(* IEC 61131-3 sources: OpenPLC-Simulator/openplc/OpenPLC/src, 47 files *)

(* ---- types.st ---- *)
(* ============================================================
   types.st — Data type definitions for the transporter simulator
   ============================================================ *)

TYPE TANK_T :
STRUCT
  tank_id    : INT;
  status     : INT;    (* NOT_USED=0, USED=1 *)
  x_position : REAL;
  y_position : REAL;
  z_position : REAL;
  stn_type   : INT;
END_STRUCT;
END_TYPE

TYPE STATION_T :
STRUCT
  tank_id       : INT;
  status        : INT;    (* NOT_USED=0, USED=1 *)
  x_position    : REAL;
  y_position    : REAL;
  z_position    : REAL;
  stn_type      : INT;    (* 0=dry, 1=wet *)
  stn_function  : INT;    (* original station type from JSON *)
  dropping_time : REAL;
  device_delay  : REAL;
END_STRUCT;
END_TYPE

TYPE PHYSICS_2D_T :
STRUCT
  x_accel_s      : REAL;
  x_decel_s      : REAL;
  x_max_mm_s     : REAL;
  z_total_mm     : REAL;
  z_slow_dry_mm  : REAL;
  z_slow_wet_mm  : REAL;
  z_slow_end_mm  : REAL;
  z_slow_mm_s    : REAL;
  z_fast_mm_s    : REAL;
  drip_delay_s   : REAL;
  avoid_mm       : REAL;
END_STRUCT;
END_TYPE

TYPE TASK_AREA_T :
STRUCT
  min_lift : INT;
  max_lift : INT;
  min_sink : INT;
  max_sink : INT;
END_STRUCT;
END_TYPE

TYPE TRANSPORTER_CFG_T :
STRUCT
  x_min_limit : REAL;
  x_max_limit : REAL;
  y_min_limit : REAL;
  y_max_limit : REAL;
  x_avoid_mm  : REAL;
  y_avoid_mm  : REAL;
  phys2d      : PHYSICS_2D_T;
  task_area   : ARRAY[1..4] OF TASK_AREA_T;
END_STRUCT;
END_TYPE

(* ── Transporter interface — production-compatible ──────────── *)
(* Used by scheduler, TWA, simulation, and production alike.     *)
(* g_transporter : ARRAY[1..TRANSPORTERS] OF STC_TRANSPORTER_T              *)
TYPE STC_TRANSPORTER_T :
STRUCT
  (* --- Command (scheduler → transporter) --- *)
  task_id            : LINT;     (* g_time_s at assignment — sync key *)
  lift_station       : INT;      (* pickup station number *)
  sink_station       : INT;      (* putdown station number *)
  treatment_time     : REAL;     (* treatment duration (s) *)
  lift_device_delay  : REAL;     (* lift station device delay (s) *)
  sink_device_delay  : REAL;     (* sink station device delay (s) *)
  dropping_time      : REAL;     (* dripping/dropping time at lift (s) *)
  (* --- Status (transporter → outside world) --- *)
  status             : INT;      (* 0=not_used 1=manual 2=half_manual 3=auto_idle 4=auto_run *)
  phase              : INT;      (* 0=idle 1=to_lift 2=lifting 3=to_sink 4=sinking *)
  running_task_id    : LINT;     (* copied from task_id when accepted *)
  current_station    : INT;      (* nearest station number *)
  remaining_time     : REAL;     (* remaining treatment time (s) *)
  (* --- Drive (runtime / TWA) --- *)
  final_target_x     : REAL;     (* destination X (station position) *)
  drive_target_x     : REAL;     (* TWA-clamped X drive target *)
  final_target_y     : REAL;     (* destination Y (3D transporter) *)
  drive_target_y     : REAL;     (* TWA-clamped Y drive target *)
  x_mm               : REAL;     (* current X position *)
  y_mm               : REAL;     (* current Y position (3D) *)
  z_mm               : REAL;     (* current Z position *)
  vel_x              : REAL;     (* X velocity *)
  z_stage            : INT;      (* Z motion sub-phase *)
  z_timer_s          : REAL;     (* Z motion timer *)
  x_min_limit        : REAL;     (* TWA lower X limit *)
  x_max_limit        : REAL;     (* TWA upper X limit *)
  (* --- General --- *)
  active             : BOOL;     (* transporter enabled *)
END_STRUCT;
END_TYPE

TYPE BATCH_T :
STRUCT
  batch_code : INT;     (* numeric batch code, e.g. 1, 2, 3 *)
  state      : INT;     (* NOT_PROCESSED=0, IN_PROCESS=1, PROCESSED=2 *)
  prog_id    : INT;     (* treatment program number *)
  cur_stage  : INT;     (* current stage number, 0 = not started *)
END_STRUCT;
END_TYPE

TYPE PROGRAM_STAGE_T :
STRUCT
  stations : ARRAY[1..5] OF INT;   (* up to MAX_PARALLELS station numbers *)
  min_time : INT;                   (* minimum processing time (seconds) *)
  max_time : INT;                   (* maximum processing time (seconds) *)
  cal_time : INT;                   (* calculated / target time (seconds) *)
END_STRUCT;
END_TYPE

TYPE TREATMENT_PROGRAM_T :
STRUCT
  program_id : INT;                      (* treatment program number *)
  stages     : ARRAY[1..30] OF PROGRAM_STAGE_T;  (* up to MAX_STAGES *)
END_STRUCT;
END_TYPE

TYPE UNIT_T :
STRUCT
  location : INT;    (* station number where unit currently is *)
  status   : INT;    (* NOT_USED=0, USED=1 *)
  state    : INT;    (* EMPTY=0, FULL=1 *)
  target   : INT;    (* TO_NONE=0, TO_LOADING=1, TO_BUFFER=2, TO_PROCESS=3, TO_UNLOAD=4, TO_AVOID=5 *)
END_STRUCT;
END_TYPE

(* ── Task Scheduler types (TSK_) ─────────────────────────────────── *)
(* Calculated batch schedule — one per unit, stages indexed 1..30       *)
(* Times are absolute epoch-offset seconds (g_time_s reference frame)   *)
(* Access: g_schedule[unit].stages[stage].entry_time                    *)

TYPE TSK_STAGE_T :
STRUCT
  station       : INT;     (* station number, 0 = unused stage *)
  entry_time    : LINT;    (* absolute arrival time (s), unix seconds *)
  exit_time     : LINT;    (* absolute departure time (s), unix seconds *)
  min_time      : REAL;    (* minimum treatment time (s) *)
  calc_time     : REAL;    (* calculated target treatment time (s) *)
  max_time      : REAL;    (* maximum treatment time (s) *)
  transfer_time : REAL;    (* transfer time from previous station (s) *)
END_STRUCT;
END_TYPE

TYPE TSK_SCHEDULE_T :
STRUCT
  stage_count : INT;                              (* number of active stages *)
  stages      : ARRAY[1..30] OF TSK_STAGE_T;     (* MAX_STAGES *)
END_STRUCT;
END_TYPE

(* Transporter task queue — indexed by transporter, then task slot       *)
(* unit is direct index to g_batches, g_programs, g_schedule, g_units   *)
(* Access: g_tasks[transporter].queue[slot].lift_station                *)

TYPE TSK_TASK_T :
STRUCT
  unit         : INT;     (* unit index 1..10, 0 = no task *)
  stage        : INT;     (* program stage that created this task *)
  lift_station : INT;     (* station to pick up from *)
  sink_station : INT;     (* station to put down to *)
  start_time   : LINT;    (* absolute time task begins (s), unix seconds *)
  finish_time  : LINT;    (* absolute time task completes (s), unix seconds *)
  calc_time    : REAL;    (* treatment calc_time for flex (s) *)
  min_time     : REAL;    (* treatment min_time for flex_down (s) *)
  max_time     : REAL;    (* treatment max_time for flex_up (s) *)
END_STRUCT;
END_TYPE

TYPE TSK_QUEUE_T :
STRUCT
  count : INT;                                    (* number of active tasks *)
  queue : ARRAY[1..10] OF TSK_TASK_T;             (* task slots, MAX_UNITS *)
END_STRUCT;
END_TYPE

(* Conflict analysis — internal working data for FB_AnalyzeConflicts    *)

TYPE TSK_CHECKED_T :
STRUCT
  unit         : INT;     (* batch unit index *)
  stage        : INT;     (* program stage *)
  transporter  : INT;     (* assigned transporter *)
  start_time   : LINT;    (* task start (s), unix seconds *)
  end_time     : LINT;    (* task end (s), unix seconds *)
  flex_down    : REAL;    (* available advance margin (s) *)
  flex_up      : REAL;    (* available delay margin (s) *)
  x_min        : REAL;    (* X-area minimum (mm) *)
  x_max        : REAL;    (* X-area maximum (mm) *)
  is_conflict  : BOOL;    (* TRUE if this task is in conflict *)
END_STRUCT;
END_TYPE

(* Precomputed movement times — timed from real motions, not calculated *)
(* Index 1..25 maps to station 101..125 (idx = stn_num - 100)           *)
(* Access: g_move[transporter].travel[from_idx].to_s[to_idx]            *)

TYPE TRAVEL_FROM_T :
STRUCT
  to_s : ARRAY[1..25] OF REAL;   (* travel time to each station (seconds) *)
END_STRUCT;
END_TYPE

TYPE MOVE_TIMES_T :
STRUCT
  lift_s  : ARRAY[1..25] OF REAL;           (* lift time per station (seconds) *)
  sink_s  : ARRAY[1..25] OF REAL;           (* sink time per station (seconds) *)
  travel  : ARRAY[1..25] OF TRAVEL_FROM_T;  (* travel[from].to_s[to] (seconds) *)
END_STRUCT;
END_TYPE

(* ── Departure Scheduler types (DEP_) ────────────────────────────── *)
(* Idle slot: a time window where a transporter has no tasks           *)
(* Used by departure scheduler to fit new batch activations            *)

TYPE DEP_IDLE_SLOT_T :
STRUCT
  start_time   : LINT;    (* idle window start (s), unix seconds *)
  end_time     : LINT;    (* idle window end (s), 0 = open-ended *)
  lift_station : INT;     (* transporter at this station at idle start *)
  sink_station : INT;     (* transporter at this station at idle end *)
END_STRUCT;
END_TYPE

TYPE DEP_IDLE_SLOT_SET_T :
STRUCT
  slots : ARRAY[1..20] OF DEP_IDLE_SLOT_T;
  count : INT;
END_STRUCT;
END_TYPE

(* Fit result: outcome of trying to fit a departure task into idle slots *)

TYPE DEP_FIT_RESULT_T :
STRUCT
  fits         : BOOL;    (* TRUE = task fits in a slot *)
  delay_s      : REAL;    (* delay needed to make it fit (s) *)
  need_extra_s : REAL;    (* extra time that does not fit (s) *)
  task_end_s   : LINT;    (* calculated task end time (s), unix seconds *)
  slot_idx     : INT;     (* index of the used idle slot *)
  trans_id     : INT;     (* transporter id that can handle it *)
END_STRUCT;
END_TYPE

(* Delay action: a schedule adjustment to accommodate departure *)

TYPE DEP_DELAY_ACTION_T :
STRUCT
  stage   : INT;     (* program stage to delay *)
  delay_s : REAL;    (* delay amount (s) *)
  target  : INT;     (* 0=batch cur_stage delay, 1=program stage delay *)
  valid   : BOOL;
END_STRUCT;
END_TYPE

(* Overlap: stations covered by multiple transporters *)

TYPE DEP_OVERLAP_T :
STRUCT
  flags : ARRAY[101..125] OF BOOL;  (* TRUE = station is in overlap zone *)
  count : INT;
END_STRUCT;
END_TYPE

(* Sandbox: isolated copy of scheduler state for departure planning *)

TYPE DEP_SANDBOX_T :
STRUCT
  schedule : ARRAY[1..10] OF TSK_SCHEDULE_T;
  batches  : ARRAY[1..10] OF BATCH_T;
  programs : ARRAY[1..10] OF TREATMENT_PROGRAM_T;
  tasks    : ARRAY[1..3] OF TSK_QUEUE_T;   (* literal — TYPE cannot use constants *)
  valid    : BOOL;
END_STRUCT;
END_TYPE

(* Pending write: data to commit from sandbox to globals after ACTIVATE *)

TYPE DEP_PENDING_WRITE_T :
STRUCT
  valid      : BOOL;
  programs   : ARRAY[1..10] OF TREATMENT_PROGRAM_T;
  schedule   : ARRAY[1..10] OF TSK_SCHEDULE_T;
  batch_unit : INT;     (* activated batch: unit index *)
  batch_stage : INT;    (* activated batch: new stage *)
  time_s     : LINT;    (* activation time (s), unix seconds *)
END_STRUCT;
END_TYPE

(* ── Calibration teaching type ─────────────────────────────────── *)
(* One per transporter. Gateway writes plan, PLC fills results.      *)
(* Only wet_station + dry_station needed: 2 normal tasks per         *)
(* transporter give all lift/sink/travel measurements.               *)
(*   Task 1: lift=dry, sink=wet → lift_dry, sink_wet, travel dry→wet *)
(*   Task 2: lift=wet, sink=dry → lift_wet, sink_dry, travel wet→dry *)
TYPE CALIBRATION_T :
STRUCT
  (* Plan — set by gateway via cfg_cmd=7 *)
  wet_station   : INT;    (* wet station number *)
  dry_station   : INT;    (* dry station number *)
  (* Results — read from g_move after MeasureMoveTimes records them *)
  lift_wet_s    : REAL;   (* lift time at wet station (s) *)
  sink_wet_s    : REAL;   (* sink time at wet station (s) *)
  lift_dry_s    : REAL;   (* lift time at dry station (s) *)
  sink_dry_s    : REAL;   (* sink time at dry station (s) *)
  x_accel_s     : REAL;   (* measured acceleration time (s) *)
  x_decel_s     : REAL;   (* measured deceleration time (s) *)
  x_max_mm_s    : REAL;   (* measured max X speed (mm/s) *)
END_STRUCT;
END_TYPE

(* ---- globals.st ---- *)
(* ============================================================
   globals.st — Global variables (shared memory + Modbus I/O)
   ============================================================ *)

VAR_GLOBAL CONSTANT
  (* ── Array size limits (used in ARRAY declarations with -a flag) ── *)
  MAX_STATIONS       : INT := 25;    (* stations 101..100+MAX_STATIONS *)
  TRANSPORTERS   : INT := 3;     (* number of transporters in this plant *)
  MAX_UNITS          : INT := 10;    (* units 1..MAX_UNITS *)
  MAX_PARALLELS      : INT := 5;     (* max parallel stations per program stage *)
  MAX_STAGES         : INT := 30;    (* max stages in a treatment program *)
  MAX_LINES          : INT := 4;     (* max production lines per transporter *)
  DEP_MAX_IDLE_SLOTS : INT := 20;    (* max idle slots per transporter *)
  DEP_MAX_DELAY_ACTS : INT := 10;    (* max delay actions per cycle *)
  DEP_MAX_WAITING    : INT := 10;    (* max waiting batches *)
  MIN_WORK_AREA      : REAL := 20.0; (* mm — TWA minimum working area *)

  (* ── Enumerated constants ── *)
  (* Unit status *)
  USED             : INT := 1;
  NOT_USED         : INT := 0;
  (* Unit state *)
  EMPTY            : INT := 0;
  FULL             : INT := 1;
  (* Unit target *)
  TO_NONE          : INT := 0;
  TO_LOADING       : INT := 1;
  TO_BUFFER        : INT := 2;
  TO_PROCESS       : INT := 3;
  TO_UNLOAD        : INT := 4;
  TO_AVOID         : INT := 5;
  (* Station type *)
  STN_DRY          : INT := 0;
  STN_WET          : INT := 1;
  (* Batch state *)
  NOT_PROCESSED    : INT := 0;
  IN_PROCESS       : INT := 1;
  PROCESSED        : INT := 2;
  (* Avoid status for stations (TWA) *)
  AVOID_NONE       : INT := 0;     (* station not avoided *)
  AVOID_PASS       : INT := 1;     (* pass through allowed, no stop *)
  AVOID_BLOCK      : INT := 2;     (* hard block, cannot pass *)
END_VAR

VAR_GLOBAL
  (* --- Shared data arrays --- *)
  g_station_count    : INT := 0;
  g_stations         : ARRAY[101..125] OF STATION_T;
  g_cfg              : ARRAY[1..TRANSPORTERS] OF TRANSPORTER_CFG_T;
  g_transporter      : ARRAY[1..TRANSPORTERS] OF STC_TRANSPORTER_T;
  g_units            : ARRAY[1..10] OF UNIT_T;
  g_batches          : ARRAY[1..10] OF BATCH_T;
  g_programs         : ARRAY[1..10] OF TREATMENT_PROGRAM_T;
  g_avoid_status     : ARRAY[101..125] OF INT;  (* AVOID_NONE/PASS/BLOCK per station *)
  g_move             : ARRAY[1..TRANSPORTERS] OF MOVE_TIMES_T;  (* precomputed movement times per transporter *)
  g_schedule         : ARRAY[1..10] OF TSK_SCHEDULE_T;  (* calculated schedule per unit *)
  g_tasks            : ARRAY[1..TRANSPORTERS] OF TSK_QUEUE_T;       (* task queue per transporter *)
  (* --- Departure Scheduler state --- *)
  g_dep_sandbox       : DEP_SANDBOX_T;                    (* sandbox: isolated copy for planning *)
  g_dep_idle_slots    : ARRAY[1..TRANSPORTERS] OF DEP_IDLE_SLOT_SET_T;  (* idle slots per transporter *)
  g_dep_waiting       : ARRAY[1..10] OF INT;              (* waiting batch unit indices *)
  g_dep_waiting_count : INT;
  g_dep_overlap       : DEP_OVERLAP_T;                    (* overlap station flags *)
  g_dep_pending       : DEP_PENDING_WRITE_T;              (* ACTIVATE → write buffer *)
  g_dep_activated     : BOOL;                             (* handshake TSK ← DEP *)
  g_dep_stable        : BOOL;                             (* handshake TSK → DEP: task list stable *)
  (* --- Calibration state --- *)
  g_cal              : ARRAY[1..TRANSPORTERS] OF CALIBRATION_T;      (* calibration plan + results per transporter *)
  g_cal_active       : BOOL;                              (* TRUE during calibration — inhibits schedulers *)
  (* --- Unix time --- *)
  (* g_time_s = absolute unix time in seconds (LINT)                       *)
  (* Gateway writes upper/lower 16-bit halves to QW160/QW161 every tick   *)
  g_time_s           : LINT;          (* absolute time in unix seconds *)
  (* --- Modbus OUTPUT: Transporter 1 (QW0..QW8) --- *)
  qw_t1_x_mm    AT %QW0  : INT;
  qw_t1_z_mm    AT %QW1  : INT;
  qw_t1_vel_x10 AT %QW2  : INT;
  qw_t1_phase   AT %QW3  : INT;
  qw_t1_z_stage AT %QW4  : INT;
  qw_t1_cur_st  AT %QW5  : INT;
  qw_t1_lift_tgt AT %QW6 : INT;
  qw_t1_sink_tgt AT %QW7 : INT;
  qw_t1_active  AT %QW8  : INT;

  (* --- Modbus OUTPUT: Transporter 2 (QW9..QW17) --- *)
  qw_t2_x_mm    AT %QW9  : INT;
  qw_t2_z_mm    AT %QW10 : INT;
  qw_t2_vel_x10 AT %QW11 : INT;
  qw_t2_phase   AT %QW12 : INT;
  qw_t2_z_stage AT %QW13 : INT;
  qw_t2_cur_st  AT %QW14 : INT;
  qw_t2_lift_tgt AT %QW15 : INT;
  qw_t2_sink_tgt AT %QW16 : INT;
  qw_t2_active  AT %QW17 : INT;

  (* --- Modbus OUTPUT: Status (QW18..QW20) --- *)
  qw_station_cnt AT %QW18 : INT;
  qw_init_done   AT %QW19 : INT;
  qw_cycle_cnt   AT %QW20 : INT;

  (* --- Modbus OUTPUT: Batch data (QW65..QW104) --- *)
  (*   10 units x 4 fields: batch_code, state, program, stage
       Unit N batch at QW65 + (N-1)*4 .. QW65 + (N-1)*4 + 3     *)
  qw_b1_code    AT %QW65  : INT;
  qw_b1_state   AT %QW66  : INT;
  qw_b1_prog    AT %QW67  : INT;
  qw_b1_stage   AT %QW68  : INT;
  qw_b2_code    AT %QW69  : INT;
  qw_b2_state   AT %QW70  : INT;
  qw_b2_prog    AT %QW71  : INT;
  qw_b2_stage   AT %QW72  : INT;
  qw_b3_code    AT %QW73  : INT;
  qw_b3_state   AT %QW74  : INT;
  qw_b3_prog    AT %QW75  : INT;
  qw_b3_stage   AT %QW76  : INT;
  qw_b4_code    AT %QW77  : INT;
  qw_b4_state   AT %QW78  : INT;
  qw_b4_prog    AT %QW79  : INT;
  qw_b4_stage   AT %QW80  : INT;
  qw_b5_code    AT %QW81  : INT;
  qw_b5_state   AT %QW82  : INT;
  qw_b5_prog    AT %QW83  : INT;
  qw_b5_stage   AT %QW84  : INT;
  qw_b6_code    AT %QW85  : INT;
  qw_b6_state   AT %QW86  : INT;
  qw_b6_prog    AT %QW87  : INT;
  qw_b6_stage   AT %QW88  : INT;
  qw_b7_code    AT %QW89  : INT;
  qw_b7_state   AT %QW90  : INT;
  qw_b7_prog    AT %QW91  : INT;
  qw_b7_stage   AT %QW92  : INT;
  qw_b8_code    AT %QW93  : INT;
  qw_b8_state   AT %QW94  : INT;
  qw_b8_prog    AT %QW95  : INT;
  qw_b8_stage   AT %QW96  : INT;
  qw_b9_code    AT %QW97  : INT;
  qw_b9_state   AT %QW98  : INT;
  qw_b9_prog    AT %QW99  : INT;
  qw_b9_stage   AT %QW100 : INT;
  qw_b10_code   AT %QW101 : INT;
  qw_b10_state  AT %QW102 : INT;
  qw_b10_prog   AT %QW103 : INT;
  qw_b10_stage  AT %QW104 : INT;

  (* --- Modbus INPUT: Commands (QW200..QW205) --- *)
  (*   NOTE: Uses %QW (holding registers) because %IW (input registers)
       are read-only from Modbus master perspective.                  *)
  iw_cmd_start_1 AT %QW200 : INT;
  iw_cmd_lift_1  AT %QW201 : INT;
  iw_cmd_sink_1  AT %QW202 : INT;
  iw_cmd_start_2 AT %QW203 : INT;
  iw_cmd_lift_2  AT %QW204 : INT;
  iw_cmd_sink_2  AT %QW205 : INT;

  (* --- Config upload protocol (QW110..QW119, QW21) --- *)
  (*   Gateway writes station config one at a time.
       Sequence number change triggers PLC processing.
       cmd=1: write_station, cmd=2: init, cmd=3: clear_all
       NOTE: Uses %QW because %IW is read-only from Modbus master.  *)
  iw_cfg_seq       AT %QW110 : INT;   (* sequence number — triggers on change *)
  iw_cfg_cmd       AT %QW111 : INT;   (* 1=write_station, 2=init, 3=clear_all *)
  iw_cfg_param     AT %QW112 : INT;   (* station_number or station_count *)
  iw_cfg_d0        AT %QW113 : INT;   (* tank_id *)
  iw_cfg_d1        AT %QW114 : INT;   (* x_position mm *)
  iw_cfg_d2        AT %QW115 : INT;   (* y_position mm *)
  iw_cfg_d3        AT %QW116 : INT;   (* z_position mm *)
  iw_cfg_d4        AT %QW117 : INT;   (* type *)
  iw_cfg_d5        AT %QW118 : INT;   (* dropping_time x10 *)
  iw_cfg_d6        AT %QW119 : INT;   (* device_delay x10 *)

  qw_cfg_ack       AT %QW21 : INT;   (* ack: last processed seq number *)

  (* --- Modbus OUTPUT: Units (QW22..QW61) --- *)
  (*   10 units x 4 fields: location, status, state, target
       Unit N at QW22 + (N-1)*4 .. QW22 + (N-1)*4 + 3            *)
  qw_u1_loc     AT %QW22 : INT;
  qw_u1_status  AT %QW23 : INT;
  qw_u1_state   AT %QW24 : INT;
  qw_u1_target  AT %QW25 : INT;
  qw_u2_loc     AT %QW26 : INT;
  qw_u2_status  AT %QW27 : INT;
  qw_u2_state   AT %QW28 : INT;
  qw_u2_target  AT %QW29 : INT;
  qw_u3_loc     AT %QW30 : INT;
  qw_u3_status  AT %QW31 : INT;
  qw_u3_state   AT %QW32 : INT;
  qw_u3_target  AT %QW33 : INT;
  qw_u4_loc     AT %QW34 : INT;
  qw_u4_status  AT %QW35 : INT;
  qw_u4_state   AT %QW36 : INT;
  qw_u4_target  AT %QW37 : INT;
  qw_u5_loc     AT %QW38 : INT;
  qw_u5_status  AT %QW39 : INT;
  qw_u5_state   AT %QW40 : INT;
  qw_u5_target  AT %QW41 : INT;
  qw_u6_loc     AT %QW42 : INT;
  qw_u6_status  AT %QW43 : INT;
  qw_u6_state   AT %QW44 : INT;
  qw_u6_target  AT %QW45 : INT;
  qw_u7_loc     AT %QW46 : INT;
  qw_u7_status  AT %QW47 : INT;
  qw_u7_state   AT %QW48 : INT;
  qw_u7_target  AT %QW49 : INT;
  qw_u8_loc     AT %QW50 : INT;
  qw_u8_status  AT %QW51 : INT;
  qw_u8_state   AT %QW52 : INT;
  qw_u8_target  AT %QW53 : INT;
  qw_u9_loc     AT %QW54 : INT;
  qw_u9_status  AT %QW55 : INT;
  qw_u9_state   AT %QW56 : INT;
  qw_u9_target  AT %QW57 : INT;
  qw_u10_loc    AT %QW58 : INT;
  qw_u10_status AT %QW59 : INT;
  qw_u10_state  AT %QW60 : INT;
  qw_u10_target AT %QW61 : INT;
  qw_unit_ack   AT %QW62 : INT;   (* ack: last processed unit write seq *)

  (* --- Modbus INPUT: Unit write command (QW120..QW125) --- *)
  (*   NOTE: Uses %QW because %IW is read-only from Modbus master.  *)
  iw_unit_seq    AT %QW120 : INT;  (* sequence — triggers on change *)
  iw_unit_id     AT %QW121 : INT;  (* unit number 1..10 *)
  iw_unit_loc    AT %QW122 : INT;  (* location (station number) *)
  iw_unit_status AT %QW123 : INT;  (* NOT_USED=0, USED=1 *)
  iw_unit_state  AT %QW124 : INT;  (* EMPTY=0, FULL=1 *)
  iw_unit_target AT %QW125 : INT;  (* TO_NONE=0, TO_LOADING=1, TO_BUFFER=2, TO_PROCESS=3, TO_UNLOAD=4, TO_AVOID=5 *)

  (* --- Modbus INPUT: Batch write protocol (QW130..QW134, ack QW63) --- *)
  (*   Writes batch data and initializes treatment program for a unit.
       PLC handler also clears all stages of g_programs[unit] on write.  *)
  iw_batch_seq     AT %QW130 : INT;  (* sequence number — triggers on change *)
  iw_batch_unit    AT %QW131 : INT;  (* unit index 1..10 *)
  iw_batch_code    AT %QW132 : INT;  (* numeric batch code *)
  iw_batch_state   AT %QW133 : INT;  (* NOT_PROCESSED=0, IN_PROCESS=1, PROCESSED=2 *)
  iw_batch_prog_id AT %QW134 : INT;  (* treatment program ID *)
  qw_batch_ack     AT %QW63  : INT;  (* ack: last processed batch write seq *)

  (* --- Modbus INPUT: Program stage write protocol (QW140..QW150, ack QW64) --- *)
  (*   Writes one treatment program stage at a time.
       Must send batch write first to set program_id and clear stages.  *)
  iw_prog_seq      AT %QW140 : INT;  (* sequence number — triggers on change *)
  iw_prog_unit     AT %QW141 : INT;  (* unit index 1..10 *)
  iw_prog_stage    AT %QW142 : INT;  (* stage index 1..30 *)
  iw_prog_s1       AT %QW143 : INT;  (* station 1 (0 = unused) *)
  iw_prog_s2       AT %QW144 : INT;  (* station 2 (0 = unused) *)
  iw_prog_s3       AT %QW145 : INT;  (* station 3 (0 = unused) *)
  iw_prog_s4       AT %QW146 : INT;  (* station 4 (0 = unused) *)
  iw_prog_s5       AT %QW147 : INT;  (* station 5 (0 = unused) *)
  iw_prog_min_time AT %QW148 : INT;  (* min processing time in seconds *)
  iw_prog_max_time AT %QW149 : INT;  (* max processing time in seconds *)
  iw_prog_cal_time AT %QW150 : INT;  (* calculated / target time in seconds *)
  qw_prog_ack      AT %QW64  : INT;  (* ack: last processed program stage seq *)

  (* --- Modbus INPUT: Unix time (QW160..QW161) --- *)
  (*   Gateway writes 32-bit unix seconds as two unsigned 16-bit halves.  *)
  (*   g_time_s = (uint16(iw_time_hi) * 65536) + uint16(iw_time_lo)      *)
  iw_time_hi   AT %QW160 : INT;  (* unix seconds upper 16 bits (unsigned) *)
  iw_time_lo   AT %QW161 : INT;  (* unix seconds lower 16 bits (unsigned) *)

  (* --- Modbus OUTPUT: Calibration status & results (QW170..QW192) --- *)
  (*   Gateway polls these during/after calibration.
       Times are × 10 for 0.1 s precision in INT Modbus registers.
       x_max is integer mm/s. *)
  qw_cal_step     AT %QW170 : INT;  (* calibration step: 0=idle, 10-40=measuring, 100=done, 200=calculating, 999=complete *)
  qw_cal_tid      AT %QW171 : INT;  (* transporter being calibrated (1..3, 0=none) *)
  (* T1 results: QW172..QW178 *)
  qw_cal_t1_lift_wet AT %QW172 : INT;
  qw_cal_t1_sink_wet AT %QW173 : INT;
  qw_cal_t1_lift_dry AT %QW174 : INT;
  qw_cal_t1_sink_dry AT %QW175 : INT;
  qw_cal_t1_x_acc    AT %QW176 : INT;
  qw_cal_t1_x_dec    AT %QW177 : INT;
  qw_cal_t1_x_max    AT %QW178 : INT;
  (* T2 results: QW179..QW185 *)
  qw_cal_t2_lift_wet AT %QW179 : INT;
  qw_cal_t2_sink_wet AT %QW180 : INT;
  qw_cal_t2_lift_dry AT %QW181 : INT;
  qw_cal_t2_sink_dry AT %QW182 : INT;
  qw_cal_t2_x_acc    AT %QW183 : INT;
  qw_cal_t2_x_dec    AT %QW184 : INT;
  qw_cal_t2_x_max    AT %QW185 : INT;
  (* T3 results: QW186..QW192 *)
  qw_cal_t3_lift_wet AT %QW186 : INT;
  qw_cal_t3_sink_wet AT %QW187 : INT;
  qw_cal_t3_lift_dry AT %QW188 : INT;
  qw_cal_t3_sink_dry AT %QW189 : INT;
  qw_cal_t3_x_acc    AT %QW190 : INT;
  qw_cal_t3_x_dec    AT %QW191 : INT;
  qw_cal_t3_x_max    AT %QW192 : INT;
END_VAR

(* ---- is_wet_station.st ---- *)
(* ============================================================
   is_wet_station.st — Check if a station type is "wet"
   ============================================================ *)

FUNCTION IsWetStationType : BOOL
VAR_INPUT
  station_type : INT;
END_VAR
  IsWetStationType := (station_type = 1) OR (station_type = 11);
END_FUNCTION

(* ---- STC_CalcHorizontalTravel.st ---- *)
(* ============================================================
   STC_CalcHorizontalTravel — Horizontal travel time (FUNCTION)
   ============================================================
   Calculates only the horizontal travel time between two stations
   (no lift/sink) using precomputed move time table.

   Converted from FUNCTION_BLOCK (STC_FB_CalcHorizontalTravel) to
   FUNCTION: the caller passes the specific transporter's
   MOVE_TIMES_T instead of using VAR_EXTERNAL g_move.

   Used by: TSK_FB_Analyze, DEP_FB_FitTaskToSlot, DEP_FB_Scheduler,
            TSK_FB_NoTreatment
   ============================================================ *)

FUNCTION STC_CalcHorizontalTravel : REAL
VAR_INPUT
  i_from_stn : INT;     (* source station number *)
  i_to_stn   : INT;     (* destination station number *)
  i_move     : MOVE_TIMES_T;   (* transporter's precomputed move times *)
END_VAR
VAR
  from_idx : INT;
  to_idx   : INT;
END_VAR

STC_CalcHorizontalTravel := 0.0;
IF i_from_stn > 0 AND i_to_stn > 0 AND i_from_stn <> i_to_stn THEN
  from_idx := i_from_stn - 100;
  to_idx   := i_to_stn - 100;
  IF from_idx >= 1 AND from_idx <= 25 AND to_idx >= 1 AND to_idx <= 25 THEN
    STC_CalcHorizontalTravel := i_move.travel[from_idx].to_s[to_idx];
  END_IF;
END_IF;

END_FUNCTION

(* ---- STC_CalcTransferTime.st ---- *)
(* ============================================================
   STC_CalcTransferTime — Total transfer time (FUNCTION)
   ============================================================
   Calculates total transfer time (lift + horizontal travel + sink)
   between two stations using precomputed move time table.

   Converted from FUNCTION_BLOCK (STC_FB_CalcTransferTime) to
   FUNCTION: the caller passes the specific transporter's
   MOVE_TIMES_T instead of using VAR_EXTERNAL g_move.

   Returns total_s only (component times lift_s/travel_s/sink_s
   are not used by any caller in the codebase).

   Used by: TSK_FB_CalcSchedule, TSK_FB_NoTreatment, DEP_FB_Scheduler
   ============================================================ *)

FUNCTION STC_CalcTransferTime : REAL
VAR_INPUT
  i_from_stn : INT;     (* source station, e.g. 105 *)
  i_to_stn   : INT;     (* destination station, e.g. 112 *)
  i_move     : MOVE_TIMES_T;   (* transporter's precomputed move times *)
END_VAR
VAR
  from_idx : INT;
  to_idx   : INT;
END_VAR

STC_CalcTransferTime := 0.0;
IF i_from_stn > 0 AND i_from_stn <> i_to_stn THEN
  from_idx := i_from_stn - 100;
  to_idx   := i_to_stn - 100;
  IF from_idx >= 1 AND from_idx <= 25 AND to_idx >= 1 AND to_idx <= 25 THEN
    STC_CalcTransferTime :=
      INT_TO_REAL(i_move.lift_s[from_idx]) / 10.0
      + INT_TO_REAL(i_move.travel[from_idx].to_s[to_idx]) / 10.0
      + INT_TO_REAL(i_move.sink_s[to_idx]) / 10.0;
  END_IF;
END_IF;

END_FUNCTION

(* ---- TWA_CalcPriority.st ---- *)
(* ============================================================
   TWA_CalcPriority.st — Priority calculation for collision avoidance

   Priority rules (from transporterWorkingArea.js):
     canEvade = FALSE  → 100000 (cannot move, others must avoid)
     phase 3 (to_sink) → 200000 + (99999 - distance_to_target)
     phase 1 (to_lift) → 100000 + (99999 - distance_to_target)
     phase 0 (idle)    → 1

   Returns REAL to avoid DINT compatibility issues.
   Values fit within REAL precision (max ~300000).
   ============================================================ *)

FUNCTION TWA_CalcPriority : REAL
VAR_INPUT
  i_phase     : INT;
  i_can_evade : BOOL;
  i_x_pos     : REAL;
  i_x_target  : REAL;
END_VAR
VAR
  dist : REAL;
END_VAR

IF NOT i_can_evade THEN
  TWA_CalcPriority := 100000.0;
  RETURN;
END_IF;

IF i_phase = 3 THEN
  dist := ABS(i_x_pos - i_x_target);
  IF dist > 99999.0 THEN dist := 99999.0; END_IF;
  TWA_CalcPriority := 200000.0 + (99999.0 - dist);
ELSIF i_phase = 1 THEN
  dist := ABS(i_x_pos - i_x_target);
  IF dist > 99999.0 THEN dist := 99999.0; END_IF;
  TWA_CalcPriority := 100000.0 + (99999.0 - dist);
ELSE
  TWA_CalcPriority := 1.0;
END_IF;

END_FUNCTION

(* ---- clear_config.st ---- *)
(* ============================================================
   clear_config.st — Clear all PLC configuration data

   Called by PLC_PRG when Gateway sends cmd=3 (clear_all).
   Zeroes out all stations, transporter configs, transporter
   states and units so the PLC is ready for fresh config upload.
   ============================================================ *)

FUNCTION_BLOCK FB_ClearConfig
VAR_EXTERNAL
  g_station_count    : INT;
  g_stations         : ARRAY[101..125] OF STATION_T;
  g_cfg              : ARRAY[1..3] OF TRANSPORTER_CFG_T;
  g_state            : ARRAY[1..3] OF TRANSPORTER_STATE_T;
  g_cmd_start        : ARRAY[1..3] OF BOOL;
  g_cmd_lift_station : ARRAY[1..3] OF INT;
  g_cmd_sink_station : ARRAY[1..3] OF INT;
  g_units            : ARRAY[1..10] OF UNIT_T;
  g_batches          : ARRAY[1..10] OF BATCH_T;
  g_programs         : ARRAY[1..10] OF TREATMENT_PROGRAM_T;
END_VAR
VAR
  i : INT;
  j : INT;
  k : INT;
END_VAR

(* --- Clear all stations --- *)
FOR i := 101 TO 125 DO
  g_stations[i].tank_id       := 0;
  g_stations[i].status        := 0;
  g_stations[i].x_position    := 0.0;
  g_stations[i].y_position    := 0.0;
  g_stations[i].z_position    := 0.0;
  g_stations[i].stn_type      := 0;
  g_stations[i].dropping_time := 0.0;
  g_stations[i].device_delay  := 0.0;
END_FOR;
g_station_count := 0;

(* --- Clear all transporter configs --- *)
FOR i := 1 TO 3 DO
  g_cfg[i].id            := 0;
  g_cfg[i].start_station := 0;
  g_cfg[i].x_min_limit   := 0.0;
  g_cfg[i].x_max_limit   := 0.0;
  g_cfg[i].phys2d.x_accel_s     := 0.0;
  g_cfg[i].phys2d.x_decel_s     := 0.0;
  g_cfg[i].phys2d.x_max_mm_s    := 0.0;
  g_cfg[i].phys2d.z_total_mm    := 0.0;
  g_cfg[i].phys2d.z_slow_dry_mm := 0.0;
  g_cfg[i].phys2d.z_slow_wet_mm := 0.0;
  g_cfg[i].phys2d.z_slow_end_mm := 0.0;
  g_cfg[i].phys2d.z_slow_mm_s   := 0.0;
  g_cfg[i].phys2d.z_fast_mm_s   := 0.0;
  g_cfg[i].phys2d.drip_delay_s  := 0.0;
  g_cfg[i].phys2d.avoid_mm      := 0.0;
END_FOR;

(* --- Clear all transporter states --- *)
FOR i := 1 TO 3 DO
  g_state[i].active              := FALSE;
  g_state[i].phase               := 0;
  g_state[i].z_stage             := 0;
  g_state[i].x_mm                := 0.0;
  g_state[i].z_mm                := 0.0;
  g_state[i].vel_x               := 0.0;
  g_state[i].vel_z               := 0.0;
  g_state[i].current_station     := 0;
  g_state[i].lift_station_target := 0;
  g_state[i].sink_station_target := 0;
  g_state[i].target_x            := 0.0;
  g_state[i].x_min_limit         := 0.0;
  g_state[i].x_max_limit         := 0.0;
  g_state[i].z_timer_s           := 0.0;
  g_cmd_start[i]        := FALSE;
  g_cmd_lift_station[i]  := 0;
  g_cmd_sink_station[i]  := 0;
END_FOR;

(* --- Clear all units --- *)
FOR i := 1 TO 10 DO
  g_units[i].location := 0;
  g_units[i].status   := 0;
  g_units[i].state    := 0;
  g_units[i].target   := 0;
END_FOR;

(* --- Clear all batches --- *)
FOR i := 1 TO 10 DO
  g_batches[i].batch_code := 0;
  g_batches[i].state      := 0;
  g_batches[i].prog_id    := 0;
  g_batches[i].cur_stage      := 0;
END_FOR;

(* --- Clear all treatment programs --- *)
FOR i := 1 TO 10 DO
  g_programs[i].program_id := 0;
  FOR j := 1 TO 30 DO
    FOR k := 1 TO 5 DO
      g_programs[i].stages[j].stations[k] := 0;
    END_FOR;
    g_programs[i].stages[j].min_time := 0;
    g_programs[i].stages[j].max_time := 0;
    g_programs[i].stages[j].cal_time := 0;
  END_FOR;
END_FOR;

END_FUNCTION_BLOCK

(* ---- DEP_FB_CalcIdleSlots.st ---- *)
(* ============================================================
   DEP_FB_CalcIdleSlots — Idle slot calculation per transporter
   ============================================================
   Calculates time windows where a transporter has no tasks.
   Each gap between consecutive tasks (or before the first /
   after the last task) is an idle slot.

   Source: transporterTaskScheduler.js calculateTransporterIdleSlots()

   Expects g_tasks[i_trans].queue to be already sorted by start_time
   (TSK_FB_Scheduler TASKS_SORT phase ensures this).

   Used by: DEP_FB_Scheduler (CHECK_ANALYZE phase)
   ============================================================ *)

FUNCTION_BLOCK DEP_FB_CalcIdleSlots
VAR_INPUT
  i_trans  : INT;      (* transporter index 1..3 *)
  i_time_s : LINT;     (* current simulation time (s), unix seconds *)
END_VAR
VAR_EXTERNAL CONSTANT
    TRANSPORTERS : INT;
END_VAR

VAR_EXTERNAL
  g_tasks          : ARRAY[1..TRANSPORTERS] OF TSK_QUEUE_T;
  g_dep_idle_slots : ARRAY[1..TRANSPORTERS] OF DEP_IDLE_SLOT_SET_T;
END_VAR
VAR
  qi       : INT;      (* queue index *)
  si       : INT;      (* slot index *)
  cnt      : INT;      (* task count for this transporter *)
  prev_end : LINT;     (* end time of previous task *)
  prev_sink : INT;     (* sink station of previous task *)
  gap_start : LINT;
  gap_end   : LINT;
  HORIZON  : LINT := 1000000000;   (* open-ended future *)
END_VAR

(* Guard *)
IF i_trans < 1 OR i_trans > 3 THEN
  RETURN;
END_IF;

(* Reset output *)
g_dep_idle_slots[i_trans].count := 0;
si := 0;
cnt := g_tasks[i_trans].count;

prev_end  := i_time_s;
prev_sink := 0;

FOR qi := 1 TO 10 DO
  IF qi > cnt THEN
    EXIT;
  END_IF;

  gap_start := prev_end;
  gap_end   := g_tasks[i_trans].queue[qi].start_time;

  (* Only create slot if there is a meaningful gap *)
  IF gap_end > gap_start + LINT#1 THEN
    si := si + 1;
    IF si <= 20 THEN
      g_dep_idle_slots[i_trans].slots[si].start_time   := gap_start;
      g_dep_idle_slots[i_trans].slots[si].end_time     := gap_end;
      g_dep_idle_slots[i_trans].slots[si].lift_station := prev_sink;
      g_dep_idle_slots[i_trans].slots[si].sink_station := g_tasks[i_trans].queue[qi].lift_station;
    END_IF;
  END_IF;

  prev_end  := g_tasks[i_trans].queue[qi].finish_time;
  prev_sink := g_tasks[i_trans].queue[qi].sink_station;
END_FOR;

(* Final slot: after last task → open-ended *)
si := si + 1;
IF si <= 20 THEN
  g_dep_idle_slots[i_trans].slots[si].start_time   := prev_end;
  g_dep_idle_slots[i_trans].slots[si].end_time     := HORIZON;
  g_dep_idle_slots[i_trans].slots[si].lift_station := prev_sink;
  g_dep_idle_slots[i_trans].slots[si].sink_station := 0;
END_IF;

g_dep_idle_slots[i_trans].count := si;

END_FUNCTION_BLOCK

(* ---- DEP_FB_CalcOverlap.st ---- *)
(* ============================================================
   DEP_FB_CalcOverlap — Overlap station detection
   ============================================================
   Identifies stations where multiple transporters can operate
   (task_area ranges overlap).  A station is marked as overlap
   if two or more different transporters have task_area ranges
   that cover it (either lift or sink range).

   Source: departureScheduler.js computeOverlapStations()

   Used by: DEP_FB_Scheduler (CALC phase)
   ============================================================ *)

FUNCTION_BLOCK DEP_FB_CalcOverlap
VAR_EXTERNAL CONSTANT
    TRANSPORTERS : INT;
END_VAR

VAR_EXTERNAL
  g_cfg         : ARRAY[1..TRANSPORTERS] OF TRANSPORTER_CFG_T;
  g_dep_overlap : DEP_OVERLAP_T;
END_VAR
VAR
  stn         : INT;
  ti          : INT;
  ai          : INT;
  cover_count : INT;
  covered     : BOOL;
  area        : TASK_AREA_T;
END_VAR

g_dep_overlap.count := 0;

FOR stn := 101 TO 125 DO
  cover_count := 0;

  FOR ti := 1 TO TRANSPORTERS DO
    covered := FALSE;
    FOR ai := 1 TO 4 DO
      IF NOT covered THEN
        area := g_cfg[ti].task_area[ai];
        (* Station is covered if within lift OR sink range *)
        IF (area.min_lift > 0 AND stn >= area.min_lift AND stn <= area.max_lift)
           OR (area.min_sink > 0 AND stn >= area.min_sink AND stn <= area.max_sink) THEN
          covered := TRUE;
        END_IF;
      END_IF;
    END_FOR;
    IF covered THEN
      cover_count := cover_count + 1;
    END_IF;
  END_FOR;

  IF cover_count >= 2 THEN
    g_dep_overlap.flags[stn] := TRUE;
    g_dep_overlap.count := g_dep_overlap.count + 1;
  ELSE
    g_dep_overlap.flags[stn] := FALSE;
  END_IF;
END_FOR;

END_FUNCTION_BLOCK

(* ---- DEP_FB_FitTaskToSlot.st ---- *)
(* ============================================================
   DEP_FB_FitTaskToSlot — Fit a departure task into idle slots
   ============================================================
   Tries to fit a single waiting-batch task into the idle slots
   of its assigned transporter.  Calculates travel times from
   the previous task's sink to this task's lift, and from this
   task's sink to the next task's lift.

   Source: transporterTaskScheduler.js fitSingleTaskToIdleSlots()

   Flex constraint: delay cannot exceed flex_up × flexUpFactor.
   If no slot fits, o_need_extra_s reports the shortfall for
   backward chaining.

   Used by: DEP_FB_Scheduler (CHECK_ANALYZE phase)
   ============================================================ *)

FUNCTION_BLOCK DEP_FB_FitTaskToSlot
VAR_INPUT
  i_lift_stn     : INT;     (* task lift station *)
  i_sink_stn     : INT;     (* task sink station *)
  i_trans_id     : INT;     (* transporter for this task *)
  i_task_start   : LINT;    (* scheduled task start time (s), unix seconds *)
  i_task_end     : LINT;    (* scheduled task end time (s), unix seconds *)
  i_shift_s      : REAL;    (* pre-applied shift (overlap delay) *)
  i_calc_time_s  : REAL;    (* treatment calc_time (s) *)
  i_max_time_s   : REAL;    (* treatment max_time (s) *)
  i_flex_factor  : REAL;    (* flex_up usage factor, e.g. 0.5 *)
  i_margin_s     : REAL;    (* minimum margin between tasks (s) *)
END_VAR
VAR_OUTPUT
  o_result : DEP_FIT_RESULT_T;
END_VAR
VAR_EXTERNAL CONSTANT
    TRANSPORTERS : INT;
END_VAR

VAR_EXTERNAL
  g_dep_idle_slots : ARRAY[1..TRANSPORTERS] OF DEP_IDLE_SLOT_SET_T;
END_VAR
VAR
  fb_travel_to   : STC_FB_CalcHorizontalTravel;
  fb_travel_from : STC_FB_CalcHorizontalTravel;
  si          : INT;
  slot_cnt    : INT;
  slot_start  : LINT;
  slot_end    : LINT;
  from_stn    : INT;    (* previous task's sink or transporter home *)
  to_stn      : INT;    (* next task's lift *)
  travel_to   : REAL;   (* travel time: prev_sink → this lift *)
  travel_from : REAL;   (* travel time: this sink → next_lift *)
  earliest    : LINT;
  latest      : LINT;
  task_dur    : LINT;
  delay       : REAL;
  flex_up     : REAL;
  capped_flex : REAL;
  best_delay  : REAL;
  best_slot   : INT;
  found       : BOOL;
END_VAR

(* Initialize output *)
o_result.fits         := FALSE;
o_result.delay_s      := 0.0;
o_result.need_extra_s := 0.0;
o_result.task_end_s   := 0;
o_result.slot_idx     := 0;
o_result.trans_id     := i_trans_id;

IF i_trans_id < 1 OR i_trans_id > 3 THEN
  RETURN;
END_IF;

task_dur   := i_task_end - i_task_start;
flex_up    := i_max_time_s - i_calc_time_s;
IF flex_up < 0.0 THEN flex_up := 0.0; END_IF;
capped_flex := flex_up * i_flex_factor;

slot_cnt   := g_dep_idle_slots[i_trans_id].count;
best_delay := 1.0E9;
best_slot  := 0;
found      := FALSE;

FOR si := 1 TO 20 DO
  IF si > slot_cnt THEN
    EXIT;
  END_IF;

  slot_start := g_dep_idle_slots[i_trans_id].slots[si].start_time;
  slot_end   := g_dep_idle_slots[i_trans_id].slots[si].end_time;

  (* ── Travel time: prev task sink → this lift ── *)
  from_stn := g_dep_idle_slots[i_trans_id].slots[si].lift_station;
  travel_to := 0.0;
  IF from_stn > 0 AND from_stn <> i_lift_stn THEN
    fb_travel_to(i_from_stn := from_stn, i_to_stn := i_lift_stn, i_trans := i_trans_id);
    travel_to := fb_travel_to.o_travel_s;
  END_IF;

  (* ── Travel time: this sink → next task lift ── *)
  to_stn := g_dep_idle_slots[i_trans_id].slots[si].sink_station;
  travel_from := 0.0;
  IF to_stn > 0 AND to_stn <> i_sink_stn THEN
    fb_travel_from(i_from_stn := i_sink_stn, i_to_stn := to_stn, i_trans := i_trans_id);
    travel_from := fb_travel_from.o_travel_s;
  END_IF;

  (* Earliest start = max(slot_start, task_start + shift) + travel_to + margin *)
  IF slot_start > (i_task_start + REAL_TO_LINT(i_shift_s)) THEN
    earliest := slot_start + REAL_TO_LINT(travel_to + i_margin_s);
  ELSE
    earliest := i_task_start + REAL_TO_LINT(i_shift_s + travel_to + i_margin_s);
  END_IF;

  (* Latest end = slot_end - travel_from - margin *)
  IF slot_end > LINT#100000000 THEN
    (* Open-ended slot *)
    latest := LINT#100000000;
  ELSE
    latest := slot_end - REAL_TO_LINT(travel_from + i_margin_s);
  END_IF;

  (* Check if task fits *)
  IF earliest + task_dur <= latest THEN
    delay := LINT_TO_REAL(earliest - i_task_start) - i_shift_s;
    IF delay < 0.0 THEN delay := 0.0; END_IF;

    (* Flex constraint: delay must not exceed capped flex *)
    IF delay <= capped_flex + i_margin_s THEN
      IF delay < best_delay THEN
        best_delay := delay;
        best_slot  := si;
        found      := TRUE;
      END_IF;
    END_IF;
  END_IF;
END_FOR;

IF found THEN
  o_result.fits      := TRUE;
  o_result.delay_s   := best_delay;
  o_result.slot_idx  := best_slot;
  o_result.task_end_s := i_task_start + REAL_TO_LINT(i_shift_s + best_delay) + task_dur;
  o_result.need_extra_s := 0.0;
ELSE
  (* Report how much extra is needed for backward chaining *)
  (* Use the best near-miss: smallest overshoot beyond capped_flex *)
  o_result.fits := FALSE;
  IF best_delay < 1.0E8 THEN
    o_result.need_extra_s := best_delay - capped_flex;
    IF o_result.need_extra_s < 0.0 THEN
      o_result.need_extra_s := 0.0;
    END_IF;
  ELSE
    o_result.need_extra_s := 0.0;  (* no slot at all *)
  END_IF;
END_IF;

END_FUNCTION_BLOCK

(* ---- DEP_FB_OverlapDelay.st ---- *)
(* ============================================================
   DEP_FB_OverlapDelay — Overlap conflict delay calculation
   ============================================================
   When a new task uses a station in the overlap zone (covered
   by multiple transporters), checks for time conflicts with
   tasks on OTHER transporters at the same station.

   Iteratively calculates the minimum delay needed to avoid
   overlap conflicts (max 20 iterations).

   Source: departureScheduler.js calculateOverlapDelay()

   Used by: DEP_FB_Scheduler / DEP_FB_FitTaskToSlot
   ============================================================ *)

FUNCTION_BLOCK DEP_FB_OverlapDelay
VAR_INPUT
  i_lift_stn   : INT;     (* task lift station *)
  i_sink_stn   : INT;     (* task sink station *)
  i_trans_id   : INT;     (* task transporter id *)
  i_task_start : LINT;    (* task start time (s), already shifted *)
  i_task_end   : LINT;    (* task end time (s), already shifted *)
  i_margin_s   : REAL;    (* conflict margin (s), default 1.0 *)
END_VAR
VAR_OUTPUT
  o_delay_s : REAL;       (* total delay needed (s), 0 = no conflict *)
END_VAR
VAR_EXTERNAL CONSTANT
    TRANSPORTERS : INT;
END_VAR

VAR_EXTERNAL
  g_tasks       : ARRAY[1..TRANSPORTERS] OF TSK_QUEUE_T;
  g_dep_overlap : DEP_OVERLAP_T;
END_VAR
VAR
  lift_is_overlap : BOOL;
  sink_is_overlap : BOOL;
  round    : INT;
  ti       : INT;    (* transporter index *)
  qi       : INT;    (* queue index *)
  max_conf : REAL;   (* maximum conflict in this round *)
  t_start  : LINT;   (* shifted task start *)
  t_end    : LINT;   (* shifted task end *)
  e_start  : LINT;   (* existing task start *)
  e_end    : LINT;   (* existing task end *)
  e_lift   : INT;
  e_sink   : INT;
  has_ovlp : BOOL;
  needed   : REAL;
END_VAR

o_delay_s := 0.0;

(* Check if lift/sink are in overlap zone *)
IF i_lift_stn >= 101 AND i_lift_stn <= 125 THEN
  lift_is_overlap := g_dep_overlap.flags[i_lift_stn];
ELSE
  lift_is_overlap := FALSE;
END_IF;
IF i_sink_stn >= 101 AND i_sink_stn <= 125 THEN
  sink_is_overlap := g_dep_overlap.flags[i_sink_stn];
ELSE
  sink_is_overlap := FALSE;
END_IF;

(* No overlap stations involved → no delay *)
IF NOT lift_is_overlap AND NOT sink_is_overlap THEN
  RETURN;
END_IF;

(* Iterative conflict resolution — max 20 rounds *)
FOR round := 1 TO 20 DO
  max_conf := 0.0;
  t_start  := i_task_start + REAL_TO_LINT(o_delay_s);
  t_end    := i_task_end + REAL_TO_LINT(o_delay_s);

  (* Check all tasks on OTHER transporters *)
  FOR ti := 1 TO TRANSPORTERS DO
    IF ti <> i_trans_id THEN
      FOR qi := 1 TO 10 DO
        IF qi > g_tasks[ti].count THEN
          EXIT;
        END_IF;

        e_lift  := g_tasks[ti].queue[qi].lift_station;
        e_sink  := g_tasks[ti].queue[qi].sink_station;
        e_start := g_tasks[ti].queue[qi].start_time;
        e_end   := g_tasks[ti].queue[qi].finish_time;

        (* Does existing task share an overlap station? *)
        has_ovlp := FALSE;
        IF lift_is_overlap AND (e_lift = i_lift_stn OR e_sink = i_lift_stn) THEN
          has_ovlp := TRUE;
        END_IF;
        IF sink_is_overlap AND (e_lift = i_sink_stn OR e_sink = i_sink_stn) THEN
          has_ovlp := TRUE;
        END_IF;

        IF has_ovlp THEN
          (* Time overlap check: task overlaps with existing? *)
          IF t_start < (e_end + REAL_TO_LINT(i_margin_s)) AND t_end > (e_start - REAL_TO_LINT(i_margin_s)) THEN
            needed := LINT_TO_REAL(e_end - t_start) + i_margin_s;
            IF needed > max_conf THEN
              max_conf := needed;
            END_IF;
          END_IF;
        END_IF;

      END_FOR;  (* qi *)
    END_IF;
  END_FOR;  (* ti *)

  (* No conflict found → done *)
  IF max_conf <= 0.0 THEN
    EXIT;
  END_IF;
  o_delay_s := o_delay_s + max_conf;
END_FOR;  (* round *)

END_FUNCTION_BLOCK

(* ---- DEP_FB_Sandbox.st ---- *)
(* ============================================================
   DEP_FB_Sandbox — Sandbox snapshot / restore / clear
   ============================================================
   Copies global scheduler state to/from the departure sandbox.
   Struct assignment `a := b` in ST copies all fields automatically.

   Source: departureScheduler.js _copyDepartureSandbox()

   Commands:
     1 = SNAPSHOT  — copy globals → g_dep_sandbox
     2 = RESTORE   — copy g_dep_sandbox → globals
     3 = CLEAR     — invalidate sandbox

   Used by: DEP_FB_Scheduler (INIT, REJECT, ACTIVATE)
   ============================================================ *)

FUNCTION_BLOCK DEP_FB_Sandbox
VAR_INPUT
  i_cmd : INT;     (* 1=SNAPSHOT, 2=RESTORE, 3=CLEAR *)
END_VAR
VAR_EXTERNAL CONSTANT
    TRANSPORTERS : INT;
END_VAR

VAR_EXTERNAL
  g_schedule    : ARRAY[1..10] OF TSK_SCHEDULE_T;
  g_batches     : ARRAY[1..10] OF BATCH_T;
  g_programs    : ARRAY[1..10] OF TREATMENT_PROGRAM_T;
  g_tasks       : ARRAY[1..TRANSPORTERS] OF TSK_QUEUE_T;
  g_dep_sandbox : DEP_SANDBOX_T;
END_VAR
VAR
  ui : INT;
  ti : INT;
END_VAR

IF i_cmd = 1 THEN
  (* ── SNAPSHOT: globals → sandbox ── *)
  FOR ui := 1 TO 10 DO
    g_dep_sandbox.schedule[ui] := g_schedule[ui];
    g_dep_sandbox.batches[ui]  := g_batches[ui];
    g_dep_sandbox.programs[ui] := g_programs[ui];
  END_FOR;
  FOR ti := 1 TO TRANSPORTERS DO
    g_dep_sandbox.tasks[ti] := g_tasks[ti];
  END_FOR;
  g_dep_sandbox.valid := TRUE;

ELSIF i_cmd = 2 THEN
  (* ── RESTORE: sandbox → globals ── *)
  IF g_dep_sandbox.valid THEN
    FOR ui := 1 TO 10 DO
      g_schedule[ui] := g_dep_sandbox.schedule[ui];
      g_batches[ui]  := g_dep_sandbox.batches[ui];
      g_programs[ui] := g_dep_sandbox.programs[ui];
    END_FOR;
    FOR ti := 1 TO TRANSPORTERS DO
      g_tasks[ti] := g_dep_sandbox.tasks[ti];
    END_FOR;
  END_IF;

ELSIF i_cmd = 3 THEN
  (* ── CLEAR: invalidate sandbox ── *)
  g_dep_sandbox.valid := FALSE;

END_IF;

END_FUNCTION_BLOCK

(* ---- DEP_FB_Scheduler.st ---- *)
(* ============================================================
   DEP_FB_Scheduler — Departure scheduler state machine
   ============================================================
   Ported from departureScheduler.js tick()

   Controls batch activation: waiting batches (stage=90) are
   checked against idle slots to see if their tasks fit into
   the existing transporter schedule without conflicts.

   Uses the "wrapper approach": works directly on globals while
   TSK is paused at phase >= 10000. Sandbox is a backup for
   rollback on REJECT.

   Phase flow:
     0      STOPPED
     1      WAIT_STABLE       (wait for TSK phase >= 10000)
     100    INIT              (snapshot, find waiting batches)
     200    CALC_OVERLAP      (compute overlap stations)
     1000   BATCH_START       (prepare current waiting batch)
     1010   CALC_SCHED        (calculate waiting batch schedule)
     1020   REBUILD_TASKS     (rebuild all task queues, sort, swap)
     1030   EXTRACT_WAIT      (extract waiting batch tasks)
     1040   CALC_IDLE         (calculate idle slots)
     2000   FIT_STAGE0        (check pickup fits in idle slot)
     2001   FIT_TASK          (check stage 1+ tasks)
     3000   APPLY_DELAY       (record delay → recalc loop)
     8000   ACTIVATE          (commit, set pending)
     8010   WAIT_SAVE         (wait for TSK to process)
     8020   END_DELAY         (stabilization ticks)
     8100   RESTART           (→ WAIT_STABLE)
     9000   REJECT            (restore sandbox, try next batch)
   ============================================================ *)

FUNCTION_BLOCK DEP_FB_Scheduler
VAR_INPUT
  i_run       : BOOL;     (* TRUE = run *)
  i_time_s    : LINT;     (* current absolute time (s), unix seconds *)
  i_tsk_phase : INT;      (* TSK_FB_Scheduler.o_phase *)
END_VAR
VAR_EXTERNAL CONSTANT
    TRANSPORTERS : INT;
END_VAR

VAR_EXTERNAL
  g_batches          : ARRAY[1..10] OF BATCH_T;
  g_units            : ARRAY[1..10] OF UNIT_T;
  g_programs         : ARRAY[1..10] OF TREATMENT_PROGRAM_T;
  g_schedule         : ARRAY[1..10] OF TSK_SCHEDULE_T;
  g_tasks            : ARRAY[1..TRANSPORTERS] OF TSK_QUEUE_T;
  g_cfg              : ARRAY[1..TRANSPORTERS] OF TRANSPORTER_CFG_T;
  g_dep_sandbox      : DEP_SANDBOX_T;
  g_dep_idle_slots   : ARRAY[1..TRANSPORTERS] OF DEP_IDLE_SLOT_SET_T;
  g_dep_overlap      : DEP_OVERLAP_T;
  g_dep_pending      : DEP_PENDING_WRITE_T;
  g_dep_activated    : BOOL;
  g_dep_stable       : BOOL;
  g_dep_waiting      : ARRAY[1..10] OF INT;
  g_dep_waiting_count : INT;
END_VAR
VAR_OUTPUT
  o_phase     : INT;
  o_wait_cnt  : INT;      (* waiting batch count *)
  o_activated : BOOL;     (* batch activated this cycle *)
END_VAR
VAR
  phase       : INT := 0;
  next_phase  : INT;

  (* ── Waiting batch management ── *)
  waiting_list  : ARRAY[1..10] OF INT;  (* unit indices with stage=90 *)
  waiting_cnt   : INT;
  cur_wait_idx  : INT;
  cur_wait_unit : INT;

  (* ── Active batch list for rebuild ── *)
  batch_list    : ARRAY[1..10] OF INT;
  batch_count   : INT;

  (* ── Extracted waiting batch tasks ── *)
  w_tasks       : ARRAY[1..30] OF TSK_TASK_T;
  w_trans       : ARRAY[1..30] OF INT;    (* transporter id per task *)
  w_task_cnt    : INT;
  cur_task_idx  : INT;

  (* ── Fit state ── *)
  fit_round      : INT;
  MAX_FIT_ROUNDS : INT := 50;
  sched_base_time : LINT;        (* adjusted base time for waiting batch *)

  (* ── Delay recording ── *)
  delay_stage  : INT;
  delay_amount : REAL;
  delay_target : INT;            (* 0=batch/stage0, 1=program stage *)

  (* ── Constants ── *)
  FLEX_FACTOR       : REAL := 0.5;
  MARGIN_S          : REAL := 5.0;
  CONFLICT_MARGIN_S : REAL := 1.0;
  MAX_INIT_WAIT_S   : REAL := 120.0;
  END_DELAY_TICKS   : INT := 100;

  (* ── End delay counter ── *)
  end_delay_cnt : INT;

  (* ── Sub-FB instances ── *)
  fb_sandbox      : DEP_FB_Sandbox;
  fb_overlap      : DEP_FB_CalcOverlap;
  fb_idle_slots   : DEP_FB_CalcIdleSlots;
  fb_fit          : DEP_FB_FitTaskToSlot;
  fb_ovlp_delay   : DEP_FB_OverlapDelay;
  fb_calc_sched   : TSK_FB_CalcSchedule;
  fb_create_tasks : TSK_FB_CreateTasks;
  fb_swap_tasks   : TSK_FB_SwapTasks;
  fb_find_trans   : STC_FB_FindTransporter;
  fb_xfer         : STC_FB_CalcTransferTime;
  fb_clear        : STC_FB_ClearTaskQueues;
  fb_sort         : STC_FB_SortTaskQueue;
  fb_collect_all  : STC_FB_CollectActiveBatches;
  fb_collect_wait : STC_FB_CollectActiveBatches;

  (* ── Temp variables ── *)
  ti : INT;  qi : INT;  bi : INT;  ui : INT;  si : INT;
  sched_trans   : INT;
  write_idx     : INT;
  loading_stn   : INT;
  first_stn     : INT;
  xfer_dur      : REAL;
  stage0_delay  : REAL;
  ovlp_delay_s  : REAL;
  total_delay_s : REAL;
  prog_idx      : INT;
  old_cal       : INT;
  new_cal       : INT;
  max_cal       : INT;
END_VAR

IF NOT i_run THEN
  phase := 0;
  o_phase := 0;
  o_activated := FALSE;
  RETURN;
END_IF;

next_phase := phase;
o_activated := FALSE;

(* ════════════════════════════════════════════════════════════ *)
(* PHASE 0: STOPPED                                           *)
(* ════════════════════════════════════════════════════════════ *)
IF phase = 0 THEN
  next_phase := 1;

(* ════════════════════════════════════════════════════════════ *)
(* PHASE 1: WAIT_STABLE                                       *)
(* Wait for TSK to be ready (phase >= 10000)                   *)
(* ════════════════════════════════════════════════════════════ *)
ELSIF phase = 1 THEN
  IF i_tsk_phase >= 10000 AND g_dep_stable THEN
    next_phase := 100;
  END_IF;

(* ════════════════════════════════════════════════════════════ *)
(* PHASE 100: INIT — snapshot sandbox, find waiting batches    *)
(* ════════════════════════════════════════════════════════════ *)
ELSIF phase = 100 THEN
  (* Snapshot globals → sandbox (backup for rollback) *)
  fb_sandbox(i_cmd := 1);

  (* Find waiting batches (cur_stage = 90) *)
  fb_collect_wait(i_mode := 1);
  waiting_cnt := fb_collect_wait.o_count;
  FOR ui := 1 TO waiting_cnt DO
    waiting_list[ui] := fb_collect_wait.o_list[ui];
  END_FOR;

  o_wait_cnt := waiting_cnt;
  g_dep_waiting_count := waiting_cnt;
  FOR ui := 1 TO waiting_cnt DO
    g_dep_waiting[ui] := waiting_list[ui];
  END_FOR;

  (* Build active batch list for rebuild phases *)
  fb_collect_all(i_mode := 0);
  batch_count := fb_collect_all.o_count;
  FOR ui := 1 TO batch_count DO
    batch_list[ui] := fb_collect_all.o_list[ui];
  END_FOR;

  IF waiting_cnt = 0 THEN
    (* No waiting batches → back to waiting *)
    fb_sandbox(i_cmd := 3);   (* clear sandbox *)
    next_phase := 1;
  ELSE
    cur_wait_idx := 1;
    next_phase := 200;
  END_IF;

(* ════════════════════════════════════════════════════════════ *)
(* PHASE 200: CALC_OVERLAP — compute overlap stations          *)
(* ════════════════════════════════════════════════════════════ *)
ELSIF phase = 200 THEN
  fb_overlap();
  next_phase := 1000;

(* ════════════════════════════════════════════════════════════ *)
(* PHASE 1000: BATCH_START — prepare current waiting batch     *)
(* ════════════════════════════════════════════════════════════ *)
ELSIF phase = 1000 THEN
  IF cur_wait_idx > waiting_cnt THEN
    (* All batches processed, none activated → back to waiting *)
    fb_sandbox(i_cmd := 2);   (* restore globals from snapshot *)
    fb_sandbox(i_cmd := 3);   (* clear sandbox *)
    next_phase := 1;
  ELSE
    cur_wait_unit := waiting_list[cur_wait_idx];
    fit_round := 0;
    sched_base_time := i_time_s;
    next_phase := 1010;
  END_IF;

(* ════════════════════════════════════════════════════════════ *)
(* PHASE 1010: CALC_SCHED — calculate waiting batch schedule   *)
(* ════════════════════════════════════════════════════════════ *)
ELSIF phase = 1010 THEN
  (* Find transporter for this batch based on its location *)
  fb_find_trans(i_lift_stn := g_units[cur_wait_unit].location, i_sink_stn := 0);
  sched_trans := fb_find_trans.o_trans_id;
  IF sched_trans = 0 THEN sched_trans := 1; END_IF;

  (* Calculate schedule using (possibly shifted) base time *)
  fb_calc_sched(
    i_unit   := cur_wait_unit,
    i_trans  := sched_trans,
    i_time_s := sched_base_time
  );

  next_phase := 1020;

(* ════════════════════════════════════════════════════════════ *)
(* PHASE 1020: REBUILD_TASKS — rebuild all task queues         *)
(* Clear, create for all active batches, sort, swap — one tick *)
(* ════════════════════════════════════════════════════════════ *)
ELSIF phase = 1020 THEN
  (* Clear all task queues *)
  fb_clear();

  (* Create tasks for ALL active batches *)
  FOR bi := 1 TO batch_count DO
    fb_create_tasks(i_unit := batch_list[bi]);
  END_FOR;

  (* Sort each queue by start_time *)
  fb_sort(i_trans := 0);

  (* Swap same-station pairs *)
  fb_swap_tasks();

  next_phase := 1030;

(* ════════════════════════════════════════════════════════════ *)
(* PHASE 1030: EXTRACT_WAIT — extract waiting batch tasks      *)
(* Copy waiting batch's tasks to w_tasks[], remove from queues *)
(* ════════════════════════════════════════════════════════════ *)
ELSIF phase = 1030 THEN
  w_task_cnt := 0;

  FOR ti := 1 TO TRANSPORTERS DO
    write_idx := 0;
    FOR qi := 1 TO g_tasks[ti].count DO
      IF g_tasks[ti].queue[qi].unit = cur_wait_unit THEN
        (* Copy to waiting task array *)
        w_task_cnt := w_task_cnt + 1;
        IF w_task_cnt <= 30 THEN
          w_tasks[w_task_cnt] := g_tasks[ti].queue[qi];
          w_trans[w_task_cnt] := ti;
        END_IF;
      ELSE
        (* Keep in queue — shift down *)
        write_idx := write_idx + 1;
        IF write_idx <> qi THEN
          g_tasks[ti].queue[write_idx] := g_tasks[ti].queue[qi];
        END_IF;
      END_IF;
    END_FOR;
    (* Clear remaining slots *)
    FOR qi := write_idx + 1 TO g_tasks[ti].count DO
      g_tasks[ti].queue[qi].unit := 0;
    END_FOR;
    g_tasks[ti].count := write_idx;
  END_FOR;

  next_phase := 1040;

(* ════════════════════════════════════════════════════════════ *)
(* PHASE 1040: CALC_IDLE — calc idle slots for all transporters*)
(* ════════════════════════════════════════════════════════════ *)
ELSIF phase = 1040 THEN
  FOR ti := 1 TO TRANSPORTERS DO
    fb_idle_slots(i_trans := ti, i_time_s := i_time_s);
  END_FOR;
  cur_task_idx := 1;
  next_phase := 2000;

(* ════════════════════════════════════════════════════════════ *)
(* PHASE 2000: FIT_STAGE0 — check pickup from loading station *)
(* Uses DEP_FB_FitTaskToSlot to fit the virtual pickup task    *)
(* ════════════════════════════════════════════════════════════ *)
ELSIF phase = 2000 THEN
  loading_stn := g_units[cur_wait_unit].location;

  (* Find first treatment station from schedule *)
  first_stn := 0;
  IF g_schedule[cur_wait_unit].stage_count >= 1 THEN
    first_stn := g_schedule[cur_wait_unit].stages[1].station;
  END_IF;

  IF first_stn = 0 OR loading_stn < 100 THEN
    (* No valid schedule or batch not on station → reject *)
    next_phase := 9000;
  ELSE
    (* Find transporter for pickup *)
    fb_find_trans(i_lift_stn := loading_stn, i_sink_stn := first_stn);
    sched_trans := fb_find_trans.o_trans_id;
    IF sched_trans = 0 THEN sched_trans := 1; END_IF;

    (* Calculate transfer time for pickup *)
    fb_xfer(i_from_stn := loading_stn, i_to_stn := first_stn, i_trans := sched_trans);
    xfer_dur := fb_xfer.o_total_s;
    IF xfer_dur < 1.0 THEN xfer_dur := 1.0; END_IF;

    (* Try fitting pickup into idle slots *)
    fb_fit(
      i_lift_stn     := loading_stn,
      i_sink_stn     := first_stn,
      i_trans_id     := sched_trans,
      i_task_start   := sched_base_time,
      i_task_end     := sched_base_time + REAL_TO_LINT(xfer_dur),
      i_shift_s      := 0.0,
      i_calc_time_s  := 0.0,
      i_max_time_s   := 2.0 * MAX_INIT_WAIT_S,
      i_flex_factor  := FLEX_FACTOR,
      i_margin_s     := MARGIN_S
    );

    IF fb_fit.o_result.fits THEN
      stage0_delay := fb_fit.o_result.delay_s;

      IF stage0_delay > MARGIN_S THEN
        (* Stage 0 needs delay — shift base time and recalculate *)
        sched_base_time := sched_base_time + REAL_TO_LINT(stage0_delay);
        fit_round := fit_round + 1;
        IF fit_round > MAX_FIT_ROUNDS THEN
          next_phase := 9000;
        ELSE
          (* Recalculate schedule with shifted base time *)
          next_phase := 1010;
        END_IF;
      ELSE
        (* Stage 0 fits → proceed to stage 1+ tasks *)
        IF w_task_cnt = 0 THEN
          next_phase := 8000;  (* No more tasks → ACTIVATE *)
        ELSE
          cur_task_idx := 1;
          next_phase := 2001;
        END_IF;
      END_IF;
    ELSE
      (* Stage 0 doesn't fit → REJECT this batch *)
      next_phase := 9000;
    END_IF;
  END_IF;

(* ════════════════════════════════════════════════════════════ *)
(* PHASE 2001: FIT_TASK — fit stage 1+ tasks one per tick      *)
(* ════════════════════════════════════════════════════════════ *)
ELSIF phase = 2001 THEN
  IF cur_task_idx > w_task_cnt THEN
    (* All tasks fit → ACTIVATE *)
    next_phase := 8000;
  ELSE
    (* Get current task data *)
    si := w_tasks[cur_task_idx].stage;
    ti := w_trans[cur_task_idx];

    (* Overlap delay check *)
    fb_ovlp_delay(
      i_lift_stn   := w_tasks[cur_task_idx].lift_station,
      i_sink_stn   := w_tasks[cur_task_idx].sink_station,
      i_trans_id   := ti,
      i_task_start := w_tasks[cur_task_idx].start_time,
      i_task_end   := w_tasks[cur_task_idx].finish_time,
      i_margin_s   := CONFLICT_MARGIN_S
    );
    ovlp_delay_s := fb_ovlp_delay.o_delay_s;

    (* Idle-slot fit check *)
    fb_fit(
      i_lift_stn     := w_tasks[cur_task_idx].lift_station,
      i_sink_stn     := w_tasks[cur_task_idx].sink_station,
      i_trans_id     := ti,
      i_task_start   := w_tasks[cur_task_idx].start_time,
      i_task_end     := w_tasks[cur_task_idx].finish_time,
      i_shift_s      := ovlp_delay_s,
      i_calc_time_s  := w_tasks[cur_task_idx].calc_time,
      i_max_time_s   := w_tasks[cur_task_idx].max_time,
      i_flex_factor  := FLEX_FACTOR,
      i_margin_s     := MARGIN_S
    );

    total_delay_s := ovlp_delay_s + fb_fit.o_result.delay_s;

    IF fb_fit.o_result.fits THEN
      IF total_delay_s <= MARGIN_S THEN
        (* Fits with negligible delay → next task *)
        cur_task_idx := cur_task_idx + 1;
        next_phase := 2001;
      ELSE
        (* Delay needed → record and recalculate *)
        delay_stage  := si;
        delay_amount := total_delay_s;
        delay_target := 1;   (* program stage *)
        next_phase   := 3000;
      END_IF;
    ELSE
      (* Does not fit → REJECT (simplified: no backward chaining) *)
      next_phase := 9000;
    END_IF;
  END_IF;

(* ════════════════════════════════════════════════════════════ *)
(* PHASE 3000: APPLY_DELAY — write delay to program, recalc   *)
(* ════════════════════════════════════════════════════════════ *)
ELSIF phase = 3000 THEN
  fit_round := fit_round + 1;
  IF fit_round > MAX_FIT_ROUNDS THEN
    next_phase := 9000;
  ELSE
    IF delay_target = 0 THEN
      (* Stage 0 delay: shift base time (handled in FIT_STAGE0, shouldn't reach here) *)
      sched_base_time := sched_base_time + REAL_TO_LINT(delay_amount);
    ELSIF delay_target = 1 THEN
      (* Program stage delay: increase cal_time *)
      prog_idx := delay_stage;
      IF prog_idx >= 1 AND prog_idx <= 30 THEN
        old_cal := g_programs[cur_wait_unit].stages[prog_idx].cal_time;
        max_cal := g_programs[cur_wait_unit].stages[prog_idx].max_time;
        new_cal := old_cal + REAL_TO_INT(delay_amount);
        IF new_cal > max_cal AND max_cal > 0 THEN
          new_cal := max_cal;
        END_IF;
        g_programs[cur_wait_unit].stages[prog_idx].cal_time := new_cal;
      END_IF;
    END_IF;
    (* Recalculate: schedule → tasks → idle → fit *)
    next_phase := 1010;
  END_IF;

(* ════════════════════════════════════════════════════════════ *)
(* PHASE 8000: ACTIVATE — commit changes to pending write      *)
(* ════════════════════════════════════════════════════════════ *)
ELSIF phase = 8000 THEN
  (* Store pending write data *)
  FOR ui := 1 TO 10 DO
    g_dep_pending.programs[ui] := g_programs[ui];
    g_dep_pending.schedule[ui] := g_schedule[ui];
  END_FOR;
  g_dep_pending.batch_unit  := cur_wait_unit;
  g_dep_pending.batch_stage := 0;    (* 90 → 0 *)
  g_dep_pending.time_s      := i_time_s;
  g_dep_pending.valid        := TRUE;

  (* Restore globals from sandbox (undo DEP's temp changes) *)
  fb_sandbox(i_cmd := 2);
  fb_sandbox(i_cmd := 3);   (* clear sandbox *)

  g_dep_activated := TRUE;
  o_activated := TRUE;

  next_phase := 8010;

(* ════════════════════════════════════════════════════════════ *)
(* PHASE 8010: WAIT_SAVE — wait for TSK to process pending     *)
(* ════════════════════════════════════════════════════════════ *)
ELSIF phase = 8010 THEN
  IF NOT g_dep_pending.valid THEN
    (* TSK has processed the pending write *)
    next_phase := 8020;
  END_IF;
  (* Otherwise keep waiting *)

(* ════════════════════════════════════════════════════════════ *)
(* PHASE 8020: END_DELAY — stabilization ticks                 *)
(* ════════════════════════════════════════════════════════════ *)
ELSIF phase = 8020 THEN
  end_delay_cnt := 0;
  next_phase := 8021;

ELSIF phase >= 8021 AND phase <= 8120 THEN
  end_delay_cnt := end_delay_cnt + 1;
  IF end_delay_cnt >= END_DELAY_TICKS THEN
    next_phase := 8100;
  ELSE
    next_phase := phase + 1;
    IF next_phase > 8120 THEN
      next_phase := 8100;
    END_IF;
  END_IF;

(* ════════════════════════════════════════════════════════════ *)
(* PHASE 8100: RESTART — back to WAIT_STABLE                   *)
(* ════════════════════════════════════════════════════════════ *)
ELSIF phase = 8100 THEN
  g_dep_activated := FALSE;
  next_phase := 1;

(* ════════════════════════════════════════════════════════════ *)
(* PHASE 9000: REJECT — restore, try next batch                *)
(* ════════════════════════════════════════════════════════════ *)
ELSIF phase = 9000 THEN
  (* Restore globals from sandbox (undo changes for this batch) *)
  fb_sandbox(i_cmd := 2);

  (* Try next waiting batch *)
  cur_wait_idx := cur_wait_idx + 1;
  IF cur_wait_idx > waiting_cnt THEN
    (* No more batches → back to waiting *)
    fb_sandbox(i_cmd := 3);
    next_phase := 1;
  ELSE
    (* Try next batch — re-snapshot is still valid *)
    next_phase := 1000;
  END_IF;

(* ════════════════════════════════════════════════════════════ *)
(* Unknown phase → reset                                       *)
(* ════════════════════════════════════════════════════════════ *)
ELSE
  next_phase := 1;
END_IF;

(* ── Phase assignment ── *)
phase := next_phase;
o_phase := phase;

END_FUNCTION_BLOCK

(* ---- fb_station_lookup.st ---- *)
(* ============================================================
   fb_station_lookup.st — Find a station by its number
   ============================================================ *)

FUNCTION_BLOCK FB_StationLookup
VAR_INPUT
  station_number : INT;
END_VAR
VAR_OUTPUT
  found           : BOOL;
  idx             : INT;
  x_mm            : REAL;
  stype           : INT;
  device_delay_s  : REAL;
  dropping_time_s : REAL;
END_VAR
VAR_EXTERNAL
  g_station_count : INT;
  g_stations      : ARRAY[1..21] OF STATION_T;
END_VAR
VAR
  i      : INT;
  tmp_st : STATION_T;
END_VAR
  found := FALSE;
  idx := 0;
  x_mm := 0.0;
  stype := 0;
  device_delay_s := 0.0;
  dropping_time_s := 0.0;

  FOR i := 1 TO g_station_count DO
    tmp_st := g_stations[i];
    IF tmp_st.number = station_number THEN
      found := TRUE;
      idx := i;
      x_mm := tmp_st.x_mm;
      stype := tmp_st.station_type;
      device_delay_s := tmp_st.device_delay_s;
      dropping_time_s := tmp_st.dropping_time_s;
      RETURN;
    END_IF;
  END_FOR;
END_FUNCTION_BLOCK

(* ---- FB_TimeMoves.st ---- *)
(* ============================================================
   FB_TimeMoves — Times actual transporter movements
   ============================================================
   Records real lift, sink, and travel times into g_move table
   by observing phase transitions in the transport cycle.
   Used by task scheduling and departure scheduling.

   Phase state machine (from plc_prg.st):
     0 → 1 : X-travel to lift station
     1 → 2 : Lift at station
     2 → 3 : X-travel to sink station
     3 → 4 : Sink at station
     4 → 0 : Cycle complete

   Filtering — only pure mechanical motion is timed:
     Travel (phase 1, 3): timer runs only when ABS(vel_x) > 0.1
       → filters out TWA collision avoidance stops.
     Lift (phase 2): timer runs only during z_stage 2, 3, 4
       → excludes device_delay + dropping_time (stage 1)
         and drip_delay (stage 5).
     Sink (phase 4): timer runs only during z_stage 7, 8
       → excludes device_delay + drip_delay (stage 6).

   Usage in plc_prg.st (one instance per transporter):
     tm1(t_id := 1, phase := g_state[1].phase,
         delta_t := 0.02, vel_x := g_state[1].vel_x,
         z_stage := g_state[1].z_stage,
         lift_stn := g_state[1].lift_station_target,
         sink_stn := g_state[1].sink_station_target,
         from_stn := g_state[1].current_station);

   Access recorded times:
     travel := g_move[1].travel[3].to_s[11];   stn 103 to 111
     lift   := g_move[1].lift_s[5];             lift at stn 105
     sink   := g_move[2].sink_s[12];            sink at stn 112
   ============================================================ *)

FUNCTION_BLOCK FB_TimeMoves
VAR_INPUT
  t_id     : INT;     (* transporter index 1..3 *)
  phase    : INT;     (* current phase 0..4 *)
  delta_t  : REAL;    (* cycle time in seconds *)
  vel_x    : REAL;    (* current X velocity mm/s *)
  z_stage  : INT;     (* current Z motion stage 0..8 *)
  lift_stn : INT;     (* lift station number, e.g. 105 *)
  sink_stn : INT;     (* sink station number, e.g. 112 *)
  from_stn : INT;     (* station before command was given *)
END_VAR
VAR
  prev_phase   : INT := -1;   (* previous phase for edge detection *)
  timer        : REAL := 0.0; (* running timer *)
  travel_from  : INT;         (* index 1..25 for travel source *)
  travel_to    : INT;         (* index 1..25 for travel destination *)
  lift_idx     : INT;         (* index 1..25 for lift station *)
  sink_idx     : INT;         (* index 1..25 for sink station *)
END_VAR
VAR_EXTERNAL
  g_move : ARRAY[1..3] OF MOVE_TIMES_T;
END_VAR

(* ---- Phase transition detection ---- *)
IF phase <> prev_phase THEN

  (* -- Save completed measurement and set up next -- *)

  IF prev_phase = 1 AND phase = 2 THEN
    (* Travel to lift complete → save travel time *)
    IF travel_from >= 1 AND travel_from <= 25
       AND travel_to >= 1 AND travel_to <= 25 THEN
      g_move[t_id].travel[travel_from].to_s[travel_to] := timer;
    END_IF;
    (* Start timing lift — timer starts at 0, accumulates only in z_stage 2-4 *)
    lift_idx := lift_stn - 100;
    timer := 0.0;

  ELSIF prev_phase = 2 AND phase = 3 THEN
    (* Lift complete → save lift time (pure mechanical Z-motion only) *)
    IF lift_idx >= 1 AND lift_idx <= 25 THEN
      g_move[t_id].lift_s[lift_idx] := timer;
    END_IF;
    (* Start timing travel to sink *)
    travel_from := lift_stn - 100;
    travel_to := sink_stn - 100;
    timer := 0.0;

  ELSIF prev_phase = 3 AND phase = 4 THEN
    (* Travel to sink complete → save travel time *)
    IF travel_from >= 1 AND travel_from <= 25
       AND travel_to >= 1 AND travel_to <= 25 THEN
      g_move[t_id].travel[travel_from].to_s[travel_to] := timer;
    END_IF;
    (* Start timing sink — timer starts at 0, accumulates only in z_stage 7-8 *)
    sink_idx := sink_stn - 100;
    timer := 0.0;

  ELSIF prev_phase = 4 AND phase = 0 THEN
    (* Sink complete → save sink time (pure mechanical Z-motion only) *)
    IF sink_idx >= 1 AND sink_idx <= 25 THEN
      g_move[t_id].sink_s[sink_idx] := timer;
    END_IF;
    timer := 0.0;

  ELSIF prev_phase = 0 AND phase = 1 THEN
    (* New cycle starting → set up travel-to-lift *)
    travel_from := from_stn - 100;
    travel_to := lift_stn - 100;
    timer := 0.0;

  ELSE
    (* Unexpected transition → just reset *)
    timer := 0.0;
  END_IF;

  prev_phase := phase;

ELSE
  (* ---- No transition: accumulate timer ---- *)

  IF phase = 1 OR phase = 3 THEN
    (* Travel: only count time when actually moving *)
    (* Filters out TWA collision avoidance stops    *)
    IF ABS(vel_x) > 0.1 THEN
      timer := timer + delta_t;
    END_IF;

  ELSIF phase = 2 THEN
    (* Lift: only mechanical Z-motion stages 2-4 *)
    (* Excludes: stage 1 (device_delay + dropping_time), stage 5 (drip_delay) *)
    IF z_stage >= 2 AND z_stage <= 4 THEN
      timer := timer + delta_t;
    END_IF;

  ELSIF phase = 4 THEN
    (* Sink: only mechanical Z-motion stages 7-8 *)
    (* Excludes: stage 6 (device_delay + drip_delay) *)
    IF z_stage >= 7 AND z_stage <= 8 THEN
      timer := timer + delta_t;
    END_IF;
  END_IF;

END_IF;

END_FUNCTION_BLOCK

(* ---- fb_xmotion.st ---- *)
(* ============================================================
   fb_xmotion.st — Horizontal motion with accel / decel
   ============================================================ *)

FUNCTION_BLOCK FB_XMotion
VAR_INPUT
  delta_t  : REAL;
  x_target : REAL;
  x_min    : REAL;
  x_max    : REAL;
  v_max    : REAL;
  t_acc    : REAL;
  t_dec    : REAL;
END_VAR
VAR_IN_OUT
  x_pos : REAL;
  v_x   : REAL;
END_VAR
VAR_OUTPUT
  arrived : BOOL;
END_VAR
VAR
  drive_target : REAL;
  distance     : REAL;
  dir          : REAL;
  a_acc        : REAL;
  a_dec        : REAL;
  brake_dist   : REAL;
  new_vel      : REAL;
  travel       : REAL;
END_VAR
  IF (x_max > x_min) THEN
    IF x_pos < x_min THEN
      drive_target := x_min;
    ELSIF x_pos > x_max THEN
      drive_target := x_max;
    ELSE
      IF x_target < x_min THEN
        drive_target := x_min;
      ELSIF x_target > x_max THEN
        drive_target := x_max;
      ELSE
        drive_target := x_target;
      END_IF;
    END_IF;
  ELSE
    drive_target := x_target;
  END_IF;

  arrived := ABS(x_pos - drive_target) <= 3.0;
  IF arrived THEN
    x_pos := drive_target;
    v_x := 0.0;
    RETURN;
  END_IF;

  IF t_acc <= 0.0 THEN t_acc := 0.001; END_IF;
  IF t_dec <= 0.0 THEN t_dec := 0.001; END_IF;
  IF v_max < 0.0 THEN v_max := 0.0; END_IF;

  a_acc := v_max / t_acc;
  a_dec := v_max / t_dec;

  dir := 1.0;
  IF drive_target < x_pos THEN
    dir := -1.0;
  END_IF;

  distance := ABS(drive_target - x_pos);

  IF a_dec > 0.0 THEN
    brake_dist := (v_x * v_x) / (2.0 * a_dec);
  ELSE
    brake_dist := 0.0;
  END_IF;

  IF brake_dist >= distance THEN
    new_vel := v_x - a_dec * delta_t;
    IF new_vel < 0.0 THEN new_vel := 0.0; END_IF;
  ELSE
    new_vel := v_x + a_acc * delta_t;
    IF new_vel > v_max THEN new_vel := v_max; END_IF;
  END_IF;

  travel := new_vel * delta_t;
  IF travel >= distance THEN
    x_pos := drive_target;
    v_x := 0.0;
    arrived := TRUE;
  ELSE
    x_pos := x_pos + dir * travel;
    v_x := new_vel;
    arrived := FALSE;
  END_IF;
END_FUNCTION_BLOCK

(* ---- SIM_FB_ClearConfig.st ---- *)
(* ============================================================
   SIM_FB_ClearConfig.st — Clear all PLC configuration data

   Called by PLC_PRG when Gateway sends cmd=3 (clear_all).
   Zeroes out all stations, transporter configs, transporter
   states and units so the PLC is ready for fresh config upload.
   ============================================================ *)

FUNCTION_BLOCK SIM_FB_ClearConfig
VAR_EXTERNAL CONSTANT
    TRANSPORTERS : INT;
END_VAR

VAR_EXTERNAL
  g_station_count    : INT;
  g_stations         : ARRAY[101..125] OF STATION_T;
  g_cfg              : ARRAY[1..TRANSPORTERS] OF TRANSPORTER_CFG_T;
  g_transporter      : ARRAY[1..TRANSPORTERS] OF STC_TRANSPORTER_T;
  g_units            : ARRAY[1..10] OF UNIT_T;
  g_batches          : ARRAY[1..10] OF BATCH_T;
  g_programs         : ARRAY[1..10] OF TREATMENT_PROGRAM_T;
  g_avoid_status     : ARRAY[101..125] OF INT;
END_VAR
VAR
  i : INT;
  j : INT;
  k : INT;
END_VAR

(* --- Clear all stations --- *)
FOR i := 101 TO 125 DO
  g_stations[i].tank_id       := 0;
  g_stations[i].status        := 0;
  g_stations[i].x_position    := 0.0;
  g_stations[i].y_position    := 0.0;
  g_stations[i].z_position    := 0.0;
  g_stations[i].stn_type      := 0;
  g_stations[i].stn_function  := 0;
  g_stations[i].dropping_time := 0.0;
  g_stations[i].device_delay  := 0.0;
END_FOR;
g_station_count := 0;

(* --- Clear all transporter configs --- *)
FOR i := 1 TO TRANSPORTERS DO
  g_cfg[i].x_min_limit   := 0.0;
  g_cfg[i].x_max_limit   := 0.0;
  g_cfg[i].y_min_limit   := 0.0;
  g_cfg[i].y_max_limit   := 0.0;
  g_cfg[i].x_avoid_mm    := 0.0;
  g_cfg[i].y_avoid_mm    := 0.0;
  g_cfg[i].phys2d.x_accel_s     := 0.0;
  g_cfg[i].phys2d.x_decel_s     := 0.0;
  g_cfg[i].phys2d.x_max_mm_s    := 0.0;
  g_cfg[i].phys2d.z_total_mm    := 0.0;
  g_cfg[i].phys2d.z_slow_dry_mm := 0.0;
  g_cfg[i].phys2d.z_slow_wet_mm := 0.0;
  g_cfg[i].phys2d.z_slow_end_mm := 0.0;
  g_cfg[i].phys2d.z_slow_mm_s   := 0.0;
  g_cfg[i].phys2d.z_fast_mm_s   := 0.0;
  g_cfg[i].phys2d.drip_delay_s  := 0.0;
  g_cfg[i].phys2d.avoid_mm      := 0.0;
  FOR j := 1 TO 4 DO
    g_cfg[i].task_area[j].min_lift := 0;
    g_cfg[i].task_area[j].max_lift := 0;
    g_cfg[i].task_area[j].min_sink := 0;
    g_cfg[i].task_area[j].max_sink := 0;
  END_FOR;
END_FOR;

(* --- Clear avoid status --- *)
FOR i := 101 TO 125 DO
  g_avoid_status[i] := 0;
END_FOR;

(* --- Clear all transporter states --- *)
FOR i := 1 TO TRANSPORTERS DO
  g_transporter[i].active          := FALSE;
  g_transporter[i].status          := 0;
  g_transporter[i].phase           := 0;
  g_transporter[i].task_id         := 0;
  g_transporter[i].running_task_id := 0;
  g_transporter[i].lift_station    := 0;
  g_transporter[i].sink_station    := 0;
  g_transporter[i].treatment_time  := 0.0;
  g_transporter[i].lift_device_delay := 0.0;
  g_transporter[i].sink_device_delay := 0.0;
  g_transporter[i].dropping_time   := 0.0;
  g_transporter[i].remaining_time  := 0.0;
  g_transporter[i].current_station := 0;
  g_transporter[i].final_target_x  := 0.0;
  g_transporter[i].drive_target_x  := 0.0;
  g_transporter[i].final_target_y  := 0.0;
  g_transporter[i].drive_target_y  := 0.0;
  g_transporter[i].x_mm            := 0.0;
  g_transporter[i].y_mm            := 0.0;
  g_transporter[i].z_mm            := 0.0;
  g_transporter[i].vel_x           := 0.0;
  g_transporter[i].z_stage         := 0;
  g_transporter[i].z_timer_s       := 0.0;
  g_transporter[i].x_min_limit     := 0.0;
  g_transporter[i].x_max_limit     := 0.0;
END_FOR;

(* --- Clear all units --- *)
FOR i := 1 TO 10 DO
  g_units[i].location := 0;
  g_units[i].status   := 0;
  g_units[i].state    := 0;
  g_units[i].target   := 0;
END_FOR;

(* --- Clear all batches --- *)
FOR i := 1 TO 10 DO
  g_batches[i].batch_code := 0;
  g_batches[i].state      := 0;
  g_batches[i].prog_id    := 0;
  g_batches[i].cur_stage      := 0;
END_FOR;

(* --- Clear all treatment programs --- *)
FOR i := 1 TO 10 DO
  g_programs[i].program_id := 0;
  FOR j := 1 TO 30 DO
    FOR k := 1 TO 5 DO
      g_programs[i].stages[j].stations[k] := 0;
    END_FOR;
    g_programs[i].stages[j].min_time := 0;
    g_programs[i].stages[j].max_time := 0;
    g_programs[i].stages[j].cal_time := 0;
  END_FOR;
END_FOR;

END_FUNCTION_BLOCK
